ABB RAPID module: TCP_mtip_on_mmtool_2.mod

MODULE TCP_mtip_on_mmtool_2
	! Points are read in order of declaration.
  ! Please do not change the order of points!

  LOCAL PERS robtarget pTCP_Point1:=[[702.2364,192.0231,768.0074],[0.00149026105646044,-0.528455138206482,-0.848959445953369,0.000890020164661109],[0,0,0,0],[9E+09,9E+09,9E+09,9E+09,9E+09,9E+09]];
	LOCAL PERS robtarget pTCP_Point2:=[[592.5673,-160.2807,642.7616],[0.0930390581488609,-0.52955037355423,-0.7869513630867,-0.302700579166412],[-1,0,0,0],[9E+09,9E+09,9E+09,9E+09,9E+09,9E+09]];
	LOCAL PERS robtarget pTCP_Point3:=[[902.0622,-23.13875,694.155],[0.236688569188118,-0.482756704092026,-0.840105891227722,-0.0717399418354034],[-1,0,0,0],[9E+09,9E+09,9E+09,9E+09,9E+09,9E+09]];
	LOCAL PERS robtarget pTCP_Point4:=[[969.8856,259.7052,705.018],[0.170421004295349,-0.465554505586624,-0.854013741016388,0.157722011208534],[0,0,0,0],[9E+09,9E+09,9E+09,9E+09,9E+09,9E+09]];
	LOCAL PERS robtarget pTCP_Point5:=[[883.9514,577.469,600.3638],[0.0183896087110043,-0.355338484048843,-0.856338202953339,0.374274283647537],[0,-1,1,0],[9E+09,9E+09,9E+09,9E+09,9E+09,9E+09]];
	LOCAL PERS robtarget pTCP_Point6:=[[537.0618,578.8711,601.8902],[0.245651736855507,0.299673765897751,0.879368662834167,-0.27669769525528],[0,-1,1,0],[9E+09,9E+09,9E+09,9E+09,9E+09,9E+09]];

ENDMODULE
